(* IEC 61131-3 sources: NMEA_parse/src, 6 files *)

(* ---- IGroup.st ---- *)
USING ControlModule;
NAMESPACE ControlSystem

    INTERFACE IGroup

    METHOD  Initialize : BOOL
        VAR_INPUT
            valve : IValve;
        END_VAR

    END_METHOD
    METHOD  Start : Int

    END_METHOD
    METHOD  Stop : Int

    END_METHOD

    METHOD  WriteCyclic
        VAR_OUTPUT
            gohome:BOOL;
            gowork:BOOL;
        END_VAR

    END_METHOD
    END_INTERFACE
END_NAMESPACE

(* ---- library.st ---- *)
USING ControlModule;
NAMESPACE ControlSystem

    CLASS PUBLIC WorkGroup
        VAR PUBLIC

        END_VAR

        VAR PRIVATE
            _valve : IValve;
        END_VAR

        METHOD PUBLIC Initialize : BOOL
            VAR_INPUT
                valve : IValve;
            END_VAR
            _valve := valve;
        END_METHOD
        METHOD PUBLIC Start : Int
            _valve.Open();
        END_METHOD
        METHOD PUBLIC Stop : Int
            _valve.Close();
        END_METHOD

        METHOD PUBLIC WriteCyclic
            VAR_OUTPUT
                gohome:BOOL;
                gowork:BOOL;
            END_VAR
            _valve.SetOutput(gohome,gowork);
        END_METHOD
    END_CLASS

END_NAMESPACE

(* ---- SubGroup.st ---- *)
USING ControlModule;

NAMESPACE ControlSystem

CLASS  SubGroup EXTENDS WorkGroup
    VAR

    END_VAR

        METHOD PUBLIC OVERRIDE Start : INT
            // 预控制逻辑
            // ....
            SUPER.Start();
        END_METHOD
END_CLASS
END_NAMESPACE

(* ---- WorkGroup.st ---- *)
USING ControlModule;
NAMESPACE ControlSystem

    CLASS PUBLIC WorkGroup IMPLEMENTS IGroup
        VAR PUBLIC

        END_VAR

        VAR PRIVATE
            _valve : IValve;
        END_VAR

        METHOD PUBLIC Initialize : BOOL
            VAR_INPUT
                valve : IValve;
            END_VAR
            _valve := valve;
        END_METHOD
        METHOD PUBLIC Start : Int
            _valve.Open();
        END_METHOD
        METHOD PUBLIC Stop : Int
            _valve.Close();
        END_METHOD

        METHOD PUBLIC WriteCyclic
            VAR_OUTPUT
                gohome:BOOL;
                gowork:BOOL;
            END_VAR
            _valve.SetOutput(gohome,gowork);
        END_METHOD
    END_CLASS

END_NAMESPACE

(* ---- configuration.st ---- *)
CONFIGURATION MyConfiguration
    TASK Main( Priority := 1);
    PROGRAM P1 WITH Main: MyProgram;

    VAR_GLOBAL
        startButton : BOOL;
        stopButton : BOOL;
        homeSignal:BOOL;
        workSignal:BOOL;
    END_VAR
END_CONFIGURATION

(* ---- program.st ---- *)
USING ControlSystem;
USING ControlModule;
PROGRAM MyProgram
    VAR_EXTERNAL
        startButton : BOOL;
        stopButton : BOOL;
        homeSignal : BOOL;
        workSignal : BOOL;
    END_VAR

    VAR
        workGroup_1 : WorkGroup;
        valve : ValveB;
        // valve : ValveB;
    END_VAR

    VAR_TEMP

    END_VAR

    workGroup_1.Initialize(valve);
    IF startButton THEN
        workGroup_1.Start();
    END_IF;
    IF stopButton THEN
        workGroup_1.Stop();
    END_IF;
    workGroup_1.WriteCyclic(gohome=>homeSignal,gowork=>workSignal);

END_PROGRAM
